# EPICS autosave request: motorApp/Db/profileMoveAxis_settings.req
$(P)$(R)M$(M)UseAxis
$(P)$(R)M$(M)Positions
